// TIA Portal V16 export
// export: Created 2024-09-05T17:39:07.2350393Z, ExportSetting WithDefaults, DisplayName Totally Integrated Automation Portal, DisplayVersion V16 Update 6, DisplayName TIA Portal Version Control Interface, DisplayVersion V16 Update 2, DisplayName TIA Portal Openness, DisplayVersion V16 Update 6, DisplayName STEP 7 Professional, DisplayVersion V16 Update 6, DisplayName STEP 7 Safety, DisplayVersion V16, DisplayName WinCC Advanced, DisplayVersion V16 Update 6
FUNCTION_BLOCK "RobotControl"   // FB15, LAD
{ S7_Optimized_Access := 'TRUE' }
VERSION : 0.1
// stored: AutoNumber true, IsIECCheckEnabled false, IsRetainMemResEnabled false, MemoryReserve 100, SetENOAutomatically false, UDAEnableTagReadback false
   VAR_INPUT
      StartReq : Bool;
      KeyExt : Bool;
      JobNrReq : Byte;
      periReady : Bool;
      stopMess : Bool;
      progAct : Bool;
      onPath : Bool;
      ext : Bool;
      internalEstop : Bool;
      home : Bool;
      pgNoReq : Bool;
      robStopped : Bool;
      jobNrBack : Byte;
   END_VAR
   VAR_OUTPUT
      StartAllowed : Bool;
      Started : Bool;
      drivesOn : Bool;
      confMess : Bool;
      ExtStart : Bool;
      moveEnable : Bool;
      reqHome : Bool;
      pgNoValid : Bool;
      reqDoor : Bool;
      jobNr : Byte;
   END_VAR
BEGIN

REGION Network 1: Possible to start external auto
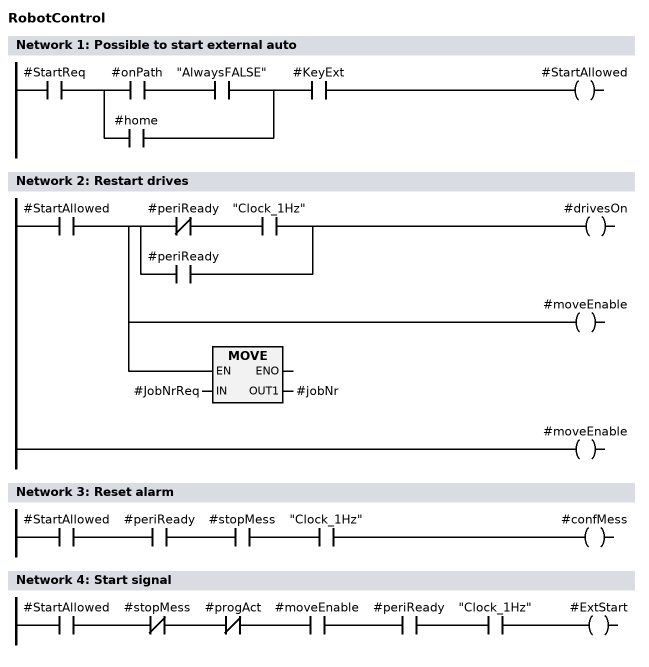
   RUNG wire#powerrail
      Contact( #StartReq )
      wire#w1
      Contact( #onPath )
      Contact( "AlwaysFALSE" )
      wire#w2
      Contact( #KeyExt )
      Coil( #StartAllowed )
   END_RUNG
   RUNG wire#w1
      Contact( #home )
   END_RUNG wire#w2
   // the same network as SCL:
   #StartAllowed := #StartReq AND ((#onPath AND "AlwaysFALSE") OR #home) AND #KeyExt;
END_REGION

REGION Network 2: Restart drives
   RUNG wire#powerrail
      Contact( #StartAllowed )
      wire#w1
      I_Contact( #periReady )
      Contact( "Clock_1Hz" )
      wire#w2
      Coil( #drivesOn )
   END_RUNG
   RUNG wire#w1
      Contact( #periReady )
   END_RUNG wire#w2
   RUNG wire#w1
      Coil( #moveEnable )
   END_RUNG
   RUNG wire#w1
      Move(in := #JobNrReq, out1 => #jobNr)
   END_RUNG
   RUNG wire#powerrail
      Coil( #moveEnable )
   END_RUNG
   // the same network as SCL:
   #drivesOn := #StartAllowed AND ((NOT #periReady AND "Clock_1Hz") OR #periReady);
   #moveEnable := #StartAllowed;
   IF #StartAllowed THEN #jobNr := #JobNrReq; END_IF;
   #moveEnable := TRUE;
END_REGION

REGION Network 3: Reset alarm
   RUNG wire#powerrail
      Contact( #StartAllowed )
      Contact( #periReady )
      Contact( #stopMess )
      Contact( "Clock_1Hz" )
      Coil( #confMess )
   END_RUNG
   // the same network as SCL:
   #confMess := #StartAllowed AND #periReady AND #stopMess AND "Clock_1Hz";
END_REGION

REGION Network 4: Start signal
   RUNG wire#powerrail
      Contact( #StartAllowed )
      I_Contact( #stopMess )
      I_Contact( #progAct )
      Contact( #moveEnable )
      Contact( #periReady )
      Contact( "Clock_1Hz" )
      Coil( #ExtStart )
   END_RUNG
   // the same network as SCL:
   #ExtStart := #StartAllowed AND NOT #stopMess AND NOT #progAct AND #moveEnable AND #periReady AND "Clock_1Hz";
END_REGION
END_FUNCTION_BLOCK
